INTERFACE I_Action

METHOD mActive : BOOL
VAR_INPUT
END_VAR
END_METHOD

METHOD mClear : BOOL
VAR_INPUT
END_VAR
END_METHOD

METHOD mCmd : BOOL
VAR_INPUT
END_VAR
END_METHOD

METHOD mComp : BOOL
VAR_INPUT
END_VAR
END_METHOD

METHOD mFault : BOOL
VAR_INPUT
END_VAR
END_METHOD

METHOD mOutput : BOOL
VAR_INPUT
END_VAR
END_METHOD

PROPERTY pActivated : BOOL
GET
END_GET
SET
END_SET
END_PROPERTY

PROPERTY pCleared : BOOL
GET
END_GET
SET
END_SET
END_PROPERTY

PROPERTY pCmdRequested : BOOL
GET
END_GET
SET
END_SET
END_PROPERTY

PROPERTY pCompleted : BOOL
GET
END_GET
SET
END_SET
END_PROPERTY

PROPERTY pFaulted : BOOL
GET
END_GET
SET
END_SET
END_PROPERTY

PROPERTY pOutputSet : BOOL
GET
END_GET
SET
END_SET
END_PROPERTY

END_INTERFACE

(* stored: Version 1.1.0.1
   Itf I_Action: Id {3db31aa2-9b0e-0f86-3751-52ce7cdd160a}
   Method mActive: Id {fcda8d2f-de47-0f0f-0f27-091c45b3c7cb}
   Method mClear: Id {f305195b-f4ad-0dcd-1dca-cd4aaf079542}
   Method mCmd: Id {3c9d666b-a006-04a1-1392-e4c094b91c0b}
   Method mComp: Id {a8eb2af8-a423-0d3d-12e4-9ab50009aa73}
   Method mFault: Id {7117549f-b8e8-0542-33ea-5bba7a21b05d}
   Method mOutput: Id {fa5e6117-12e2-0635-328b-5a2e0a6cc282}
   Property pActivated: Id {04711a7d-b419-07b4-244f-8ae065f71bfb}
   Get Get: Id {90ecb2f7-c5e1-0808-0757-1f231f43a225}
   Set Set: Id {b43a13f9-d84e-0191-20d7-df485d85d941}
   Property pCleared: Id {daafbe19-b0b8-099d-0233-c4697b914c04}
   Get Get: Id {c0f192bd-4dd1-0091-3936-41484b80f3fb}
   Set Set: Id {60b57e4c-95d7-0a31-152f-edfabd449752}
   Property pCmdRequested: Id {e03e11e9-6098-070f-21b3-7d2d5f505d6e}
   Get Get: Id {fc2fad2c-a112-067e-1112-b0ef2ae2349f}
   Set Set: Id {9d7cb77c-99c9-0aa5-0ef8-1d73189c3361}
   Property pCompleted: Id {c321b6e1-9d8a-01fa-121a-2c471ad46cec}
   Get Get: Id {48e725cb-8a2b-0d88-3512-bebc1805397e}
   Set Set: Id {ada5ba1a-ac75-057d-0261-3a6d6bec1c08}
   Property pFaulted: Id {76118985-4cae-07ad-195d-27c907a5aa0a}
   Get Get: Id {f85d5bb0-c7ea-0fda-1bea-81a5b9a20809}
   Set Set: Id {ee239b15-fd3c-0a9d-1c21-78cf431bfb60}
   Property pOutputSet: Id {415afdf0-50c1-0c46-14a1-b6a86da7db50}
   Get Get: Id {87c3d8b5-06eb-0e5a-314f-92a3b88e80d0}
   Set Set: Id {63679e65-0f31-0c7b-0a9e-37633a6e593b} *)
